(* PLC project Generated.project, CODESYS CODESYS V3.5 SP19 Patch 1 *)
(* stored: creationDateTime 2026-09-06T13:00:42.561324, modificationDateTime 2026-09-06T13:00:42.561324 *)

(* ═══════════════════════════════════════════════════════════════ ST_BypassSync — Bypass de la surveillance synchronisation M1/M2 🔒 Doctrine : actionnable UNIQUEMENT en MAINT_N2, RETAIN, jamais masque les autres défauts du même bloc (voir REGISTRE_ACTIONS_Bypass_v1.0 (archive)). ═══════════════════════════════════════════════════════════════ *)
TYPE ST_BypassSync : STRUCT
  Global : BOOL := FALSE;  (* 🌐 Bypass GLOBAL synchro : ignore toute erreur de synchronisation *)
  Initialized : BOOL := FALSE;  (* 🚦 flag restauration boot *)
END_STRUCT;
END_TYPE
